FUNCTION_BLOCK Q_ActiveMask_AUI (* Command change active mask with AUI adapter (UINT) *)
  (* Standard: ISO 11783-6; Description: Copyright (c) 2026 Meisterschulen am Ostbahnhof This program and the accompanying materials are made available under the terms of the Eclipse Public License 2.0 which is available at https://www.eclipse.org/legal/epl-2.0/ SPDX-License-Identifier: EPL-2.0 *)
  (* Version 1.0, 2026-09-10, Franz Höpfinger, Meisterschulen am Ostbahnhof, AUI adapter wrapper for Q_ActiveMask *)
  PACKAGE isobus::UT::Q;
  (* Documentation:
  Command change active mask with AUI adapter ( Part 6 - F.34 )
   This FB is an AUI adapter wrapper around Q_ActiveMask.
  *)
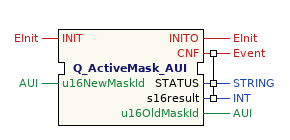
  EVENT_INPUT
    INIT : EInit; (* Service Initialization *)
  END_EVENT
  EVENT_OUTPUT
    INITO : EInit; (* Initialization Confirm *)
    CNF WITH STATUS, s16result; (* Confirmation of Requested Service *)
  END_EVENT
  VAR_OUTPUT
    STATUS : STRING; (* Service Status *)
    s16result : INT; (* retval see description *)
  END_VAR
  SOCKETS
    u16NewMaskId : adapter::types::unidirectional::AUI; (* New active mask ID *)
  END_SOCKETS
  PLUGS
    u16OldMaskId : adapter::types::unidirectional::AUI; (* Old active mask ID *)
  END_PLUGS
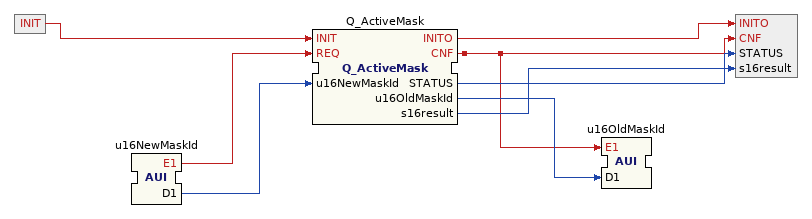
  FBS
    Q_ActiveMask : isobus::UT::Q::Q_ActiveMask;
  END_FBS
  EVENT_CONNECTIONS
    INIT TO Q_ActiveMask.INIT;
    Q_ActiveMask.INITO TO INITO;
    Q_ActiveMask.CNF TO CNF;
    u16NewMaskId.E1 TO Q_ActiveMask.REQ;
    Q_ActiveMask.CNF TO u16OldMaskId.E1;
  END_CONNECTIONS
  DATA_CONNECTIONS
    Q_ActiveMask.STATUS TO STATUS;
    u16NewMaskId.D1 TO Q_ActiveMask.u16NewMaskId;
    Q_ActiveMask.u16OldMaskId TO u16OldMaskId.D1;
    Q_ActiveMask.s16result TO s16result;
  END_CONNECTIONS
END_FUNCTION_BLOCK
